// TIA Portal V16 export
// export: Created 2021-11-12T13:33:04.1527238Z, ExportSetting WithDefaults, DisplayName Totally Integrated Automation Portal, DisplayVersion V16 Update 3, DisplayName TIA Portal Version Control Interface, DisplayVersion V16 Update 2, DisplayName TIA Portal Openness, DisplayVersion V16 Update 3, DisplayName SINAMICS Startdrive Advanced, DisplayVersion V16 Update 5, DisplayName SINAMICS Startdrive G130, G150, S120, S150, SINAMICS MV, S210, DisplayVersion V16 Update 5, DisplayName SINAMICS Startdrive G110M, G120, G120C, G120D, G120P, G115D, DisplayVersion V16 Update 5, DisplayName STEP 7 Professional, DisplayVersion V16 Update 3, DisplayName STEP 7 Safety, DisplayVersion V16, DisplayName WinCC UA Professional, DisplayVersion V16 Update 3
DATA_BLOCK "IDB_StationTHM2"   // DB67
VERSION : 0.1
// stored: AutoNumber true, DBAccessibleFromOPCUA true, InstanceOfName StationTHM2, InstanceOfType FB
"StationTHM2"
   // VAR_INPUT
   //    IS_Inputs : "UDT_COMM_THM1_CRS";
   // END_VAR
   // VAR_OUTPUT
   //    OS_Outputs : "UDT_COMM_CRS_THM1";
   //    OS_Specific : "UDT_THM_Status_specific";
   // END_VAR
   // VAR
   //    SF_Alarm1 : "STD_DI_Mon";
   //    SF_Alarm2 : "STD_DI_Mon";
   //    SF_Alarm3 : "STD_DI_Mon";
   //    SF_Alarm4 : "STD_DI_Mon";
   //    SF_Alarm5 : "STD_DI_Mon";
   //    SF_Alarm6 : "STD_DI_Mon";
   //    SF_Alarm7 : "STD_DI_Mon";
   //    SF_Alarm8 : "STD_DI_Mon";
   //    SS_Edge : Array[0..15] of Bool;
   //    SS_ParamTemp : Struct
   //       PartType : Int;
   //       ConvSpd : Int;
   //    END_STRUCT;
   //    SB1ParamChanged : Bool;
   // END_VAR
BEGIN
END_DATA_BLOCK
